FUNCTION_BLOCK LDateAndTimePointerComparer EXTENDS Object IMPLEMENTS IPointerComparer
VAR
	_ClassName : STRING := __POUNAME();
END_VAR

{attribute 'monitoring' := 'call'}
PROPERTY ClassName : STRING
GET
ClassName := _ClassName;
END_GET
END_PROPERTY

{attribute "object_name" := "Compare"}
METHOD Compare : COMPARISION_RESULT
VAR_INPUT
	left : PVOID;
	right : PVOID;
END_VAR
VAR
	leftPointer : POINTER TO LDATE_AND_TIME; 
	rightPointer : POINTER TO LDATE_AND_TIME; 
END_VAR
IF left = 0 AND right = 0 THEN
	Compare := COMPARISION_RESULT.FIRST_EQUAL_TO_SECOND;
	RETURN;
END_IF

IF left = 0 THEN
	Compare := COMPARISION_RESULT.FIRST_LESS_THAN_SECOND;
	RETURN;	
END_IF

IF right = 0 THEN
	Compare := COMPARISION_RESULT.FIRST_GREATER_THAN_SECOND;
	RETURN;	
END_IF

leftPointer := left;
rightPointer := right;

IF leftPointer^ < rightPointer^ THEN
	Compare := COMPARISION_RESULT.FIRST_LESS_THAN_SECOND;
ELSIF leftPointer^ > rightPointer^ THEN
	Compare := COMPARISION_RESULT.FIRST_GREATER_THAN_SECOND;
ELSE
	Compare := COMPARISION_RESULT.FIRST_EQUAL_TO_SECOND;	
END_IF
END_METHOD

{attribute 'monitoring' := 'call'}
PROPERTY Size : ULINT
GET
Size := XSIZEOF(THIS^);
END_GET
END_PROPERTY

END_FUNCTION_BLOCK

(* stored: Version 1.1.0.1
   POU LDateAndTimePointerComparer: Id {e25fe3ad-49bc-420a-9880-625ed94683f7}, SpecialFunc None
   Property ClassName: Id {7a0f8760-2f5b-43d3-9a7c-25b1b735888d}
   Get Get: Id {5768412f-5255-4e17-8c9d-1bbcc8cd5ba5}
   Method Compare: Id {2f6f0996-e0c5-4cbe-a45c-bee661589f7d}
   Property Size: Id {44a203bf-62d1-428e-b472-9acaf7918f7b}
   Get Get: Id {a226199e-66c5-4a5c-91ca-0fb261ab03df} *)
